(* CODESYS project IRTopdracht.project

Project tree, tasks and I/O mapping:
  Device : CODESYS Control Win V3 x64, 3S - Smart Software Solutions GmbH, version 3.5.11.40
    application Application
      libraries: Standard, * (System)
      task MainTask (cyclic, interval t#20ms, priority 1) calls PLC_PRG
      task VISU_TASK (cyclic, interval 100 ms, priority 31) calls VisuElems.Visu_Prg
      program PLC_PRG [ST]
      global variables Tank
      visualisation Visualization
      function block PID [ST]
      Symbols
      function block CalcD [ST]
      function block CalcI [ST]
  libraries: VisuSymbols, 3.5.10.0 (System)
  text list GlobalTextList
*)

// Device/Application/Tank
{attribute 'qualified_only'}
VAR_GLOBAL
	VALVE_FILL		:	REAL; // 0 - 10
	VALVE_DISCHARGE	:	REAL; // 0 - 10
	
	METER_FLOW		:	REAL; // 0 - 10
	METER_LEVEL		:	REAL; // 0 - 10
END_VAR

// Device/Application/PLC_PRG
PROGRAM PLC_PRG
VAR
	pid				:	PID;
	
	Lmin			:	REAL := -2;
	Lmax			:	REAL := 2;
	setPoint		:	REAL := 5.0;
	
	kP				:	REAL := 1.5;
	kI				:	REAL := 0.1;
	kD				:	REAL := 2.5;
END_VAR

pid(KP := kP, KI := kI, KD := kD, IlimMin := Lmin, IlimMax := Lmax, setpoint := setpoint, in := Tank.METER_LEVEL);

IF pid.Y > 0 THEN
	Tank.VALVE_FILL := pid.Y;
	Tank.VALVE_DISCHARGE := 0;
ELSIF pid.Y < 0 THEN
	Tank.VALVE_DISCHARGE := (pid.Y * -1);	
	Tank.VALVE_FILL := 0;
ELSE
	Tank.VALVE_DISCHARGE := 0;
	Tank.VALVE_FILL := 0;
END_IF

END_PROGRAM

// Device/Application/PID
FUNCTION_BLOCK PID
VAR_INPUT
	KP	:	REAL;
	KI	:	REAL;
	KD	:	REAL;
	
	
	IlimMin		:	REAL; // Lower limit of the integrator
	IlimMax		:	REAL; // Upper limit of the integrator
	setPoint	:	REAL;
	in			:	REAL;
END_VAR
VAR_OUTPUT
	limt		:	BOOL; // Limit of the PID (active/inactive)
	Y			:	REAL; // Output of the PID
END_VAR
VAR
	Dcalc		:	CalcD;
	Icalc		:	CalcI;
	
	error		:	REAL;
END_VAR

error := setPoint - in;
Icalc(input := in, KI := KI, outMin := IlimMin, outMax := IlimMax, error := error);	
Dcalc(input := in, KD := KD, error := error);

Y := KP * error + Icalc.output + Dcalc.output;

END_FUNCTION_BLOCK

// Device/Application/CalcD
FUNCTION_BLOCK CalcD
VAR_INPUT
	input			:	REAL; // inputvalue
	KD				:	REAL;
	error			:	REAL;
END_VAR
VAR_OUTPUT
	output			:	REAL;
END_VAR
VAR
	init			:	BOOL;
	currentTime		:	DWORD;
	lastTime		: 	DWORD;
	timeDiff 		: 	REAL;
	lastError		:	REAL;
END_VAR

currentTime := TIME_TO_DWORD(TIME());
timeDiff := DWORD_TO_REAL(currentTime - lastTime); // Calculate the timedifference between now and last time 

IF NOT init THEN // Only calculate the old value if it's the first time the differentiatior is running.
	init := TRUE; 
	lastError := error;
ELSIF timeDiff > 0.0 THEN
	output := KD * ((error - lastError) / timeDiff);
	lastError := error;
ELSE
	output := 0.0;
END_IF
lastTime := currentTime;

END_FUNCTION_BLOCK

// Device/Application/CalcI
FUNCTION_BLOCK CalcI
VAR_INPUT
	input		:	REAL;
	KI			:	REAL;
	outMin		:	REAL; // Minimum outputvalue
	outMax		:	REAL; // Maximum outputvalue
	error		:	REAL;
END_VAR
VAR_OUTPUT
	limt		:	BOOL;
	output		:	REAL;
END_VAR
VAR	
	oldValue	:	REAL;
	init		:	BOOL;
	currentTime	: 	DWORD;
	lastTime	: 	DWORD;
	timeDiff	: 	REAL;
	
	errorSum	:	REAL;
END_VAR

currentTime := TIME_TO_DWORD(TIME()); // to seconds
timeDiff := DWORD_TO_REAL(currentTime - lastTime); // Calculate the timedifference between now and last time 
// Integrator calculations
IF NOT init THEN
	init := TRUE;
	oldValue := input;
ELSIF timeDiff > 0.0 THEN
	errorSum := errorSum + (error * timeDiff);
	output := KI * errorSum;
END_IF
//END_IF

IF output >= outMax THEN
	//output := outMax;
	errorSum := outMax * (1/KI);
	limt := TRUE;
ELSIF output <= outMin THEN
	output := outMin;
	errorSum := outMin * (1/KI);
	limt := TRUE;
ELSE
	limt := FALSE;
END_IF

lastTime := currentTime;

END_FUNCTION_BLOCK

// Device/Application/Visualization
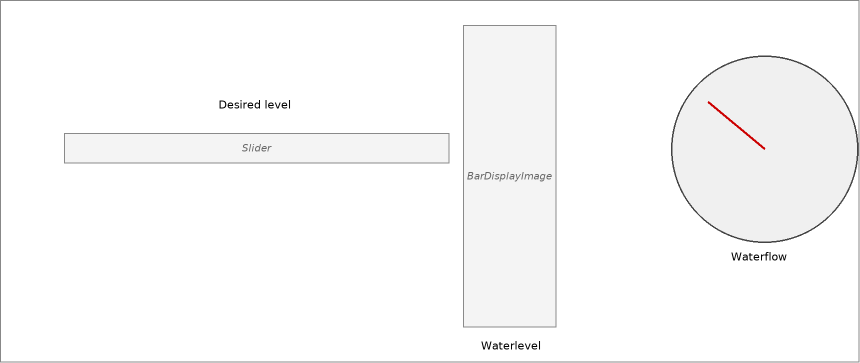
VISUALIZATION Visualization  // 860x363
    Label (180,90 150x30), "Desired level"
    Meter90 (671,45 187x208), value: Tank.METER_FLOW, style: Meter-Meter90-Gray, scale format: %.1f, scale 0..10
    Label (436,331 150x30), "Waterlevel"
    Label (684,242 150x30), "Waterflow"
    BarDisplayImage (463,25 93x302), value: Tank.METER_LEVEL, style: BarDisplayImage-Gray, scale format: %.1f, scale 0..10
    Slider (64,133 385x30), variable: PLC_PRG.setPoint, scale 0..10
END_VISUALIZATION
